(* IEC 61131-3 sources: Std_PalletMover/Class/I_PivotWheel, 1 file *)

(* ---- I_PivotWheel.st ---- *)
(*!
<Class
	Name               = "I_PivotWheel"
	Revision           = "0.0"
	RealtimeTask       = "false"
	CyclicTask         = "false"
	BackgroundTask     = "false"
	Sigmatek           = "false"
	OSInterface        = "false"
	HighPriority       = "false"
	Automatic          = "false"
	UpdateMode         = "Prescan"
	SharedCommandTable = "true"
	Objectsize         = "(750,300)">
	<Channels>
		<Server Name="ClassSvr" Visualized="false" Initialize="false" WriteProtected="true" Retentive="false"/>
		<Server Name="DistanceToCenterX" Visualized="false" Initialize="true" WriteProtected="false" Retentive="File" Comment="There is a coordinate frame attached to the center of the AGV. This sever describes the position of the wheel in this coordinate frame in mm. This is the x-component."/>
		<Server Name="DistanceToCenterY" Visualized="false" Initialize="true" WriteProtected="false" Retentive="File" Comment="There is a coordinate frame attached to the center of the AGV. This sever describes the position of the wheel in this coordinate frame in mm. This is the y-component."/>
		<Server Name="PivotWheelReferenced" Visualized="false" Initialize="false" WriteProtected="true" Retentive="false"/>
		<Client Name="objDrive" Required="false" Internal="false"/>
		<Client Name="objSteer" Required="false" Internal="false"/>
	</Channels>
</Class>
*)
I_PivotWheel : CLASS
	TYPE
#pragma pack(push, 1)
	  tPivotWheelParameters : STRUCT  //! <Type Public="true" Name="tPivotWheelParameters"/>
	    pwp_DistanceToCenterX : REAL;
	    pwp_DistanceToCenterY : REAL;
	    pwp_PivotWheelReferenced : DINT;
	  END_STRUCT;
#pragma pack(pop)
#pragma pack(push, 4)
	  tPivotWheelStatus : STRUCT  //! <Type Public="true" Name="tPivotWheelStatus"/>
	    pws_PivotWheelExists : BOOL;
	    pws_Driving : HandleSteering::tDriveStatus;
	    pws_Steering : HandleSteering::tDriveStatus;
	  END_STRUCT;
#pragma pack(pop)
	END_TYPE
  //Servers:
	ClassSvr 	: SvrChCmd_DINT;
	DistanceToCenterX 	: SvrCh_REAL;
	DistanceToCenterY 	: SvrCh_REAL;
	PivotWheelReferenced 	: SvrCh_DINT;
  //Clients:
	objSteer 	: CltChCmd_HandleSteering;
	objDrive 	: CltChCmd_HandleSteering;
  //Variables:
  //Functions:

	FUNCTION GLOBAL SendCurrentState;

	FUNCTION GLOBAL GetPivotWheelParameters
		VAR_OUTPUT
			returnValue 	: tPivotWheelParameters;
		END_VAR;

	FUNCTION GLOBAL SetPivotWheelSetpoints
		VAR_INPUT
			SPSpeed 	: REAL;
			SPAngle 	: REAL;
		END_VAR;

	FUNCTION GLOBAL GetActualAngle
		VAR_OUTPUT
			returnValue 	: REAL;
		END_VAR;

	FUNCTION GLOBAL GetActualSpeed
		VAR_OUTPUT
			returnValue 	: REAL;
		END_VAR;

	FUNCTION GLOBAL GetPivotWheelStatus
		VAR_OUTPUT
			returnValue 	: tPivotWheelStatus;
		END_VAR;

	FUNCTION VIRTUAL GLOBAL PivotWheelReferenced::Read
		VAR_OUTPUT
			output (EAX) 	: DINT;
		END_VAR;
  //Tables:
	FUNCTION @STD
		VAR_OUTPUT
			ret_code	: CONFSTATES;
		END_VAR;
	FUNCTION GLOBAL TAB @CT_;
END_CLASS;

#pragma usingLtd HandleSteering

FUNCTION GLOBAL I_PivotWheel::SendCurrentState

END_FUNCTION

FUNCTION GLOBAL I_PivotWheel::GetPivotWheelParameters
	VAR_OUTPUT
		returnValue 	: tPivotWheelParameters;
	END_VAR

  returnValue.pwp_DistanceToCenterX := DistanceToCenterX;
  returnValue.pwp_DistanceToCenterY := DistanceToCenterY;
  returnValue.pwp_PivotWheelReferenced := PivotWheelReferenced;

END_FUNCTION

FUNCTION GLOBAL I_PivotWheel::SetPivotWheelSetpoints
	VAR_INPUT
		SPSpeed 	: REAL;
		SPAngle 	: REAL;
	END_VAR

  objDrive.Setpoint.Write(SPSpeed);
  objSteer.Setpoint.Write(SPAngle);

END_FUNCTION

FUNCTION VIRTUAL GLOBAL I_PivotWheel::PivotWheelReferenced::Read
	VAR_OUTPUT
		output (EAX) 	: DINT;
	END_VAR

  PivotWheelReferenced := objDrive.GetReferenced() & objSteer.GetReferenced();
	output := PivotWheelReferenced;

END_FUNCTION

FUNCTION GLOBAL I_PivotWheel::GetActualAngle
	VAR_OUTPUT
		returnValue 	: REAL;
	END_VAR
  VAR
  	tmpDriveStatus : HandleSteering::tDriveStatus;
  END_VAR

  tmpDriveStatus := objSteer.GetDriveStatus();
  returnValue := tmpDriveStatus.ds_Actual;

END_FUNCTION

FUNCTION GLOBAL I_PivotWheel::GetActualSpeed
	VAR_OUTPUT
		returnValue 	: REAL;
	END_VAR
  VAR
  	tmpDriveStatus : HandleSteering::tDriveStatus;
  END_VAR

  tmpDriveStatus := objDrive.GetDriveStatus();
  returnValue := tmpDriveStatus.ds_Actual;

END_FUNCTION

FUNCTION GLOBAL I_PivotWheel::GetPivotWheelStatus
	VAR_OUTPUT
		returnValue 	: tPivotWheelStatus;
	END_VAR

  returnValue.pws_PivotWheelExists := TRUE;
  returnValue.pws_Driving := objDrive.GetDriveStatus();
  returnValue.pws_Steering := objSteer.GetDriveStatus();

END_FUNCTION
